Staubli VAL3: pp.pjx

--- pp.pjx ---
Parameters version=s7.1 stackSize=5000 millimeterUnit=true
Program file=Pick.pgx
Program file=Place.pgx
Program file=RobotMotion.pgx
Program file=start.pgx
Program file=stop.pgx
Program file=User.pgx
Data file=pp.dtx

--- pp.dtx ---
bool bBool1 = true
jointRx jHome
mdesc mNomSpeed
mdesc mSlow = {accel=25, vel=25, decel=25, tmax=25, rmax=25}
num nRep
pointRx pPointrx1[3]
  [0] = {x=611.54, y=-334.812005, z=260.499354, rx=-4.959689, ry=154.036634, rz=-5.509255, fatherId=world[0]}
  [1] = {x=739.655424, y=-22.141465, z=103.226279, rx=9.330921, ry=168.093288, rz=-33.667519, fatherId=world[0]}
  [2] = {x=330.134697, y=799.531714, z=-139.574889, rx=170.585193, ry=-7.909797, rz=71.354806, fatherId=world[0]}
tool tTool1 = {fatherId=flange[0], ioLink=valve1}
screen Interfaz
num nPact[2]
num nPdes[2]
bool bBool2 = true

--- start.pgx ---
program start()
begin
  call RobotMotion()
end

--- Pick.pgx ---
program Pick(pointRx pPos (dimensions=1))
begin
  movel(appro(pPos,{0,0,-50,0,0,0}),tTool1,mNomSpeed)
  delay(3)
  open(tTool1)
  movel(pPos,tTool1,mSlow)
  delay(3)
  close(tTool1)
  movel(appro(pPos,{0,0,-50,0,0,0}),tTool1,mSlow)
  delay(3)
end

--- Place.pgx ---
program Place(pointRx pPos (dimensions=1))
begin
  movel(appro(pPos,{0,0,-50,0,0,0}),tTool1,mNomSpeed)
  delay(3)
  movel(appro(pPos,{0,0,-1,0,0,0}),tTool1,mSlow)
  delay(3)
  open(tTool1)
  movel(appro(pPos,{0,0,-50,0,0,0}),tTool1,mSlow)
  delay(3)
  close(tTool1)
end

--- RobotMotion.pgx ---
program RobotMotion()
begin
  movej(jHome,tTool1,mNomSpeed)
  delay(3)
  while (bBool1)
    call Pick(pPointrx1[nRep])
    nRep=nRep+1

    if nRep==3
      nRep=0
      //bBool1.false
    endIf
    call Place(pPointrx1[nRep])
  endWhile
end

--- User.pgx ---
program User()
  local num nMenu
  local pointRx pPos
begin
  userPage()
  while ()
    cls(Interfaz)
    title(Interfaz,"Pick-and-Place")
    nMenu = getKey()
    switch nmenu
      case 271
        pPos = pPointrx1[0]
      break
      case 272
        pPos = pPointrx1[1]
      break
      case 273
        pPos = pPointrx1[2]
      break
      default
        pPos=jHome
      break
    endSwitch
    if bBool2==true
      call Pick(pPos)
    else
      call Place(pPos)
    bBool2=bBool2!
  endWhile
end
